// Mitsubishi GX Developer project: 01-CODE   PLC: FX1N

PROGRAM MAIN
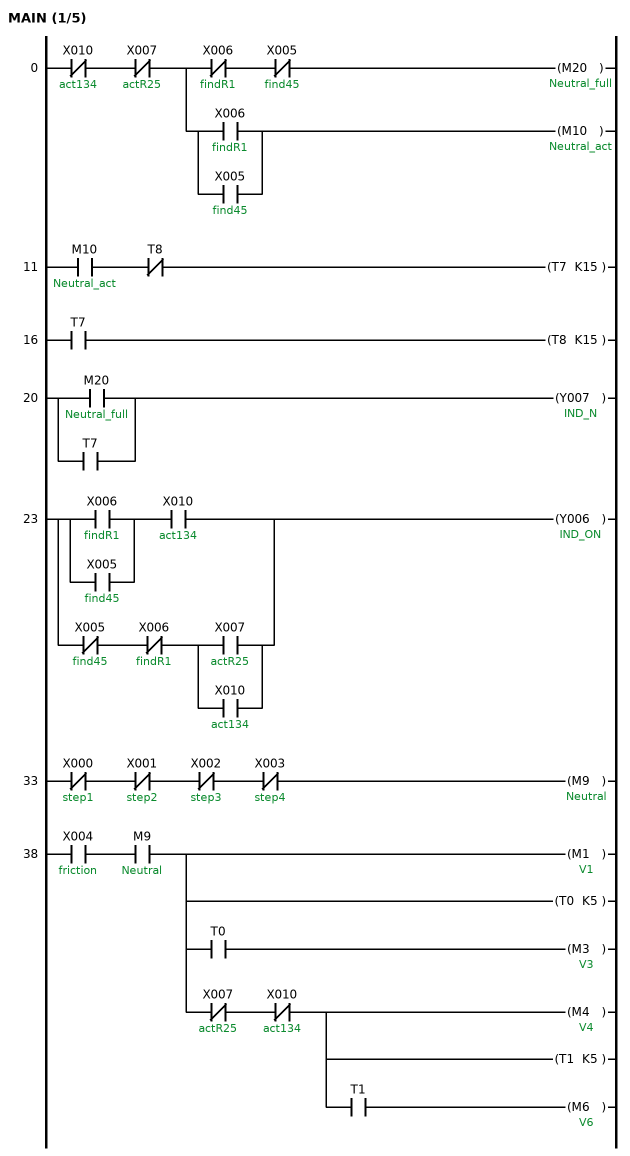
0     LDI     X010  ; act134
      ANI     X007  ; actR25
      MPS
      ANI     X006  ; findR1
      ANI     X005  ; find45
      OUT     M20  ; Neutral_full
      MPP
      LD      X006  ; findR1
      OR      X005  ; find45
      ANB
      OUT     M10  ; Neutral_act
11    LD      M10  ; Neutral_act
      ANI     T8
      OUT     T7 K15
16    LD      T7
      OUT     T8 K15
20    LD      M20  ; Neutral_full
      OR      T7
      OUT     Y007  ; IND_N
23    LD      X006  ; findR1
      OR      X005  ; find45
      AND     X010  ; act134
      LDI     X005  ; find45
      ANI     X006  ; findR1
      LD      X007  ; actR25
      OR      X010  ; act134
      ANB
      ORB
      OUT     Y006  ; IND_ON
33    LDI     X000  ; step1
      ANI     X001  ; step2
      ANI     X002  ; step3
      ANI     X003  ; step4
      OUT     M9  ; Neutral
38    LD      X004  ; friction
      AND     M9  ; Neutral
      OUT     M1  ; V1
      OUT     T0 K5
      MPS
      AND     T0
      OUT     M3  ; V3
      MPP
      ANI     X007  ; actR25
      ANI     X010  ; act134
      OUT     M4  ; V4
      OUT     T1 K5
      AND     T1
      OUT     M6  ; V6
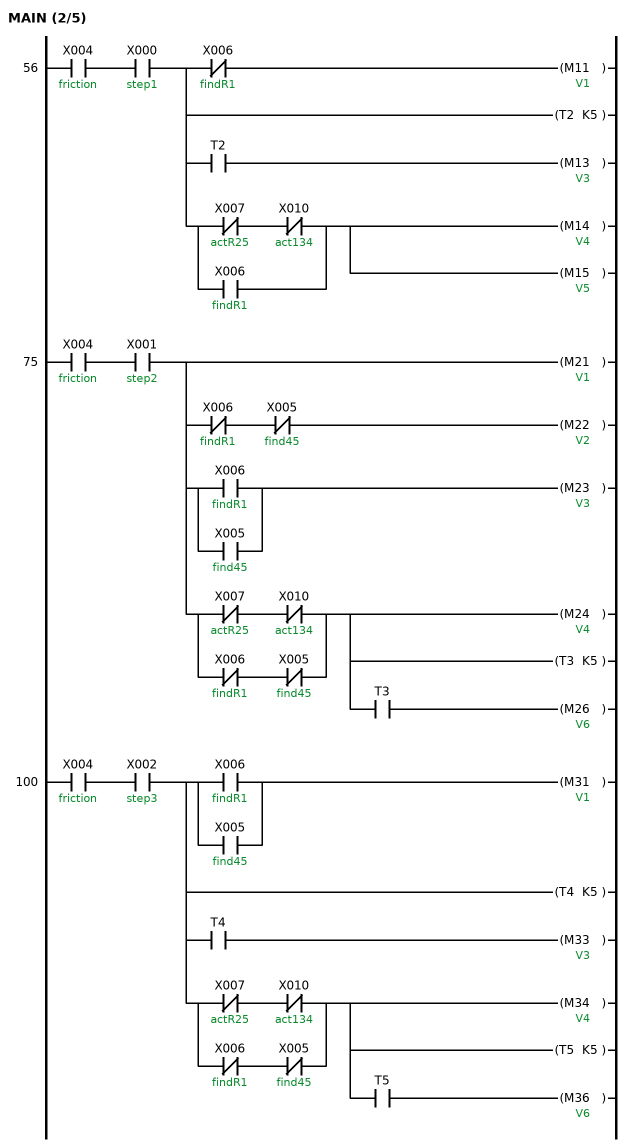
56    LD      X004  ; friction
      AND     X000  ; step1
      MPS
      ANI     X006  ; findR1
      OUT     M11  ; V1
      MPP
      OUT     T2 K5
      MPS
      AND     T2
      OUT     M13  ; V3
      MPP
      LDI     X007  ; actR25
      ANI     X010  ; act134
      OR      X006  ; findR1
      ANB
      OUT     M14  ; V4
      OUT     M15  ; V5
75    LD      X004  ; friction
      AND     X001  ; step2
      OUT     M21  ; V1
      MPS
      ANI     X006  ; findR1
      ANI     X005  ; find45
      OUT     M22  ; V2
      MRD
      LD      X006  ; findR1
      OR      X005  ; find45
      ANB
      OUT     M23  ; V3
      MPP
      LDI     X007  ; actR25
      ANI     X010  ; act134
      LDI     X006  ; findR1
      ANI     X005  ; find45
      ORB
      ANB
      OUT     M24  ; V4
      OUT     T3 K5
      AND     T3
      OUT     M26  ; V6
100   LD      X004  ; friction
      AND     X002  ; step3
      MPS
      LD      X006  ; findR1
      OR      X005  ; find45
      ANB
      OUT     M31  ; V1
      MPP
      OUT     T4 K5
      MPS
      AND     T4
      OUT     M33  ; V3
      MPP
      LDI     X007  ; actR25
      ANI     X010  ; act134
      LDI     X006  ; findR1
      ANI     X005  ; find45
      ORB
      ANB
      OUT     M34  ; V4
      OUT     T5 K5
      AND     T5
      OUT     M36  ; V6
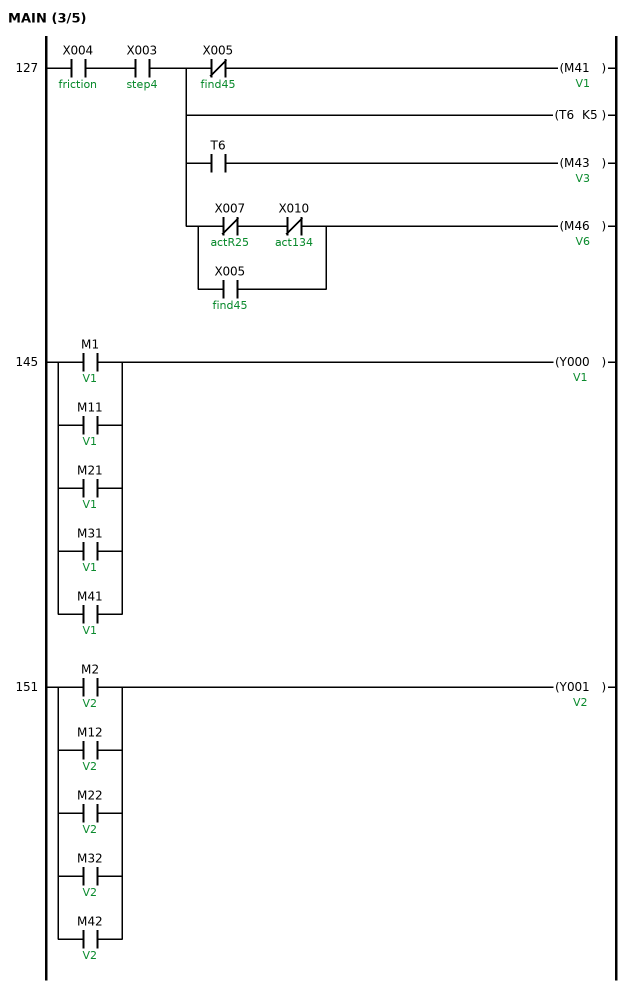
127   LD      X004  ; friction
      AND     X003  ; step4
      MPS
      ANI     X005  ; find45
      OUT     M41  ; V1
      MPP
      OUT     T6 K5
      MPS
      AND     T6
      OUT     M43  ; V3
      MPP
      LDI     X007  ; actR25
      ANI     X010  ; act134
      OR      X005  ; find45
      ANB
      OUT     M46  ; V6
145   LD      M1  ; V1
      OR      M11  ; V1
      OR      M21  ; V1
      OR      M31  ; V1
      OR      M41  ; V1
      OUT     Y000  ; V1
151   LD      M2  ; V2
      OR      M12  ; V2
      OR      M22  ; V2
      OR      M32  ; V2
      OR      M42  ; V2
      OUT     Y001  ; V2
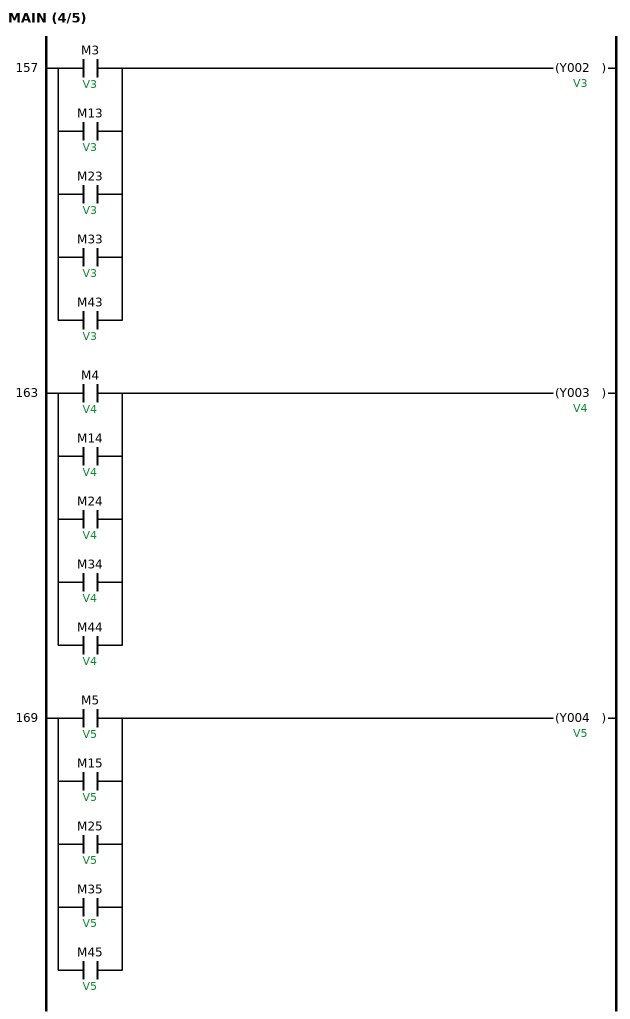
157   LD      M3  ; V3
      OR      M13  ; V3
      OR      M23  ; V3
      OR      M33  ; V3
      OR      M43  ; V3
      OUT     Y002  ; V3
163   LD      M4  ; V4
      OR      M14  ; V4
      OR      M24  ; V4
      OR      M34  ; V4
      OR      M44  ; V4
      OUT     Y003  ; V4
169   LD      M5  ; V5
      OR      M15  ; V5
      OR      M25  ; V5
      OR      M35  ; V5
      OR      M45  ; V5
      OUT     Y004  ; V5
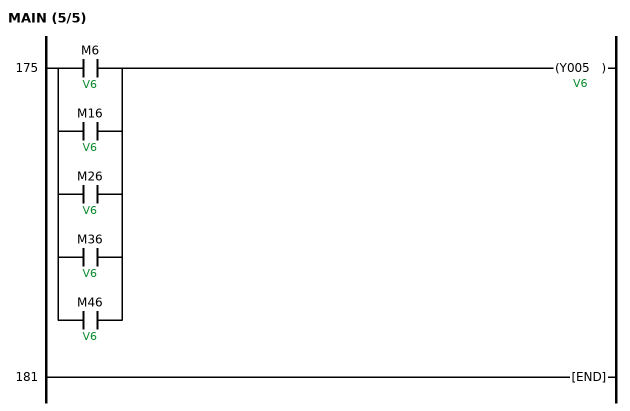
175   LD      M6  ; V6
      OR      M16  ; V6
      OR      M26  ; V6
      OR      M36  ; V6
      OR      M46  ; V6
      OUT     Y005  ; V6
181   END
END_PROGRAM
